(* CoDeSys 2.3 library: TcBase2.lib *)
(* Libraries: STANDARD.LIB 5.6.98 11:03:02 *)

(* Data type *)
TYPE FW_ULINT :
STRUCT
	loUDINT : UDINT;
	hiUDINT : UDINT;
END_STRUCT
END_TYPE

(* POU FW_GetActualDcTime2, ST *)
FUNCTION FW_GetActualDcTime2 : UDINT
VAR_INPUT
	p: POINTER TO FW_ULINT;
END_VAR
VAR
END_VAR
;
END_FUNCTION

(* POU FW_GetCurDcTaskTime2, ST *)
FUNCTION FW_GetCurDcTaskTime2 : UDINT
VAR_INPUT
	p: POINTER TO FW_ULINT;
END_VAR
VAR
END_VAR
;
END_FUNCTION

(* POU FW_GetCurDcTickTime2, ST *)
FUNCTION FW_GetCurDcTickTime2 : UDINT
VAR_INPUT
	p: POINTER TO FW_ULINT;
END_VAR
VAR
END_VAR
;
END_FUNCTION

(* POU FW_GetCurTaskSystemTime2, ST *)
FUNCTION FW_GetCurTaskSystemTime2 : UDINT
VAR_INPUT
	p: POINTER TO FW_ULINT;
END_VAR
VAR
END_VAR
;
END_FUNCTION
